TYPE E_DisconnectorFault :
(
    NONE := 0,                  // Arıza yok
    THERMAL := 1,               // Termik arıza
    CONTACTOR_ON := 2,          // ON kontaktör geri bildirim hatası
    CONTACTOR_OFF := 3,         // OFF kontaktör geri bildirim hatası
    MOTION_TIMEOUT := 4,        // Hareket zaman aşımı
    BOTH_LIMITS := 5,           // Her iki limit aktif
    INTERLOCK := 6,             // Toprak bıçağı interlock hatası
    EARTH_SWITCH := 7           // Toprak bıçağı senkronizasyon hatası
);
END_TYPE

(* stored: Version 1.1.0.1, ProductVersion 3.1.4024.15
   EnumerationTextList E_DisconnectorFault: Id {8941a61c-7cdd-4082-90a5-807e4cf2989b} *)
